PROGRAM P_MotionControl
VAR
	fbJoystick 				: FB_Joystick;
	fbGetStartPos 			: FB_StartPos;
	fbWinchVelIntegrator 	: FB_Integrator;
	fWinchVelRef 			: LREAL;
	fWinchPosRef 			: LREAL;
	fWinchPos 				: LREAL;
	fInitialWinchPos 		: LREAL;
	bWinchVelIntegratorOn	: BOOL := TRUE; 
	bAutoEnable 			: BOOL;
	bManualEnable 			: BOOL;
	fWinchPosRefManual 		: LREAL;
	fWinchVelRefManual 		: LREAL;
	fWinchVelRefAuto 		: LREAL;
END_VAR

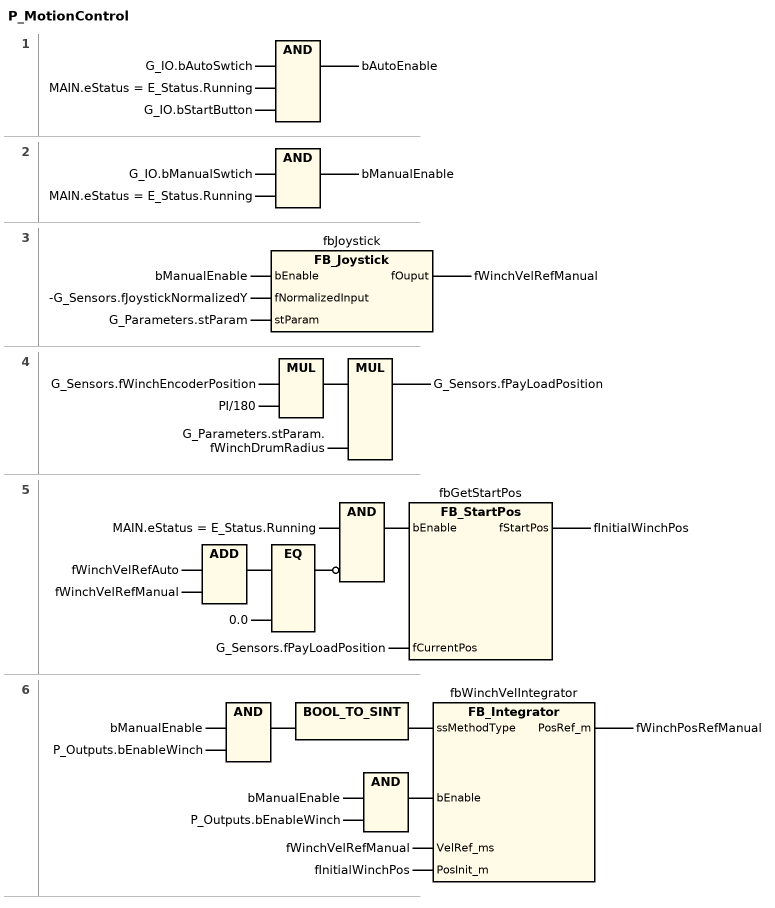
// NETWORK 1
bAutoEnable := G_IO.bAutoSwtich AND (MAIN.eStatus = E_Status.Running) AND G_IO.bStartButton;

// NETWORK 2
bManualEnable := G_IO.bManualSwtich AND (MAIN.eStatus = E_Status.Running);

// NETWORK 3
fbJoystick(
    bEnable := bManualEnable,
    fNormalizedInput := -G_Sensors.fJoystickNormalizedY,
    stParam := G_Parameters.stParam); // FB_Joystick
fWinchVelRefManual := fbJoystick.fOuput;

// NETWORK 4
G_Sensors.fPayLoadPosition := (G_Sensors.fWinchEncoderPosition * (PI/180)) * G_Parameters.stParam.fWinchDrumRadius;

// NETWORK 5
fbGetStartPos(bEnable := (MAIN.eStatus = E_Status.Running) AND NOT (fWinchVelRefAuto + fWinchVelRefManual = 0.0), fCurrentPos := G_Sensors.fPayLoadPosition); // FB_StartPos
fInitialWinchPos := fbGetStartPos.fStartPos;

// NETWORK 6
fbWinchVelIntegrator(
    ssMethodType := BOOL_TO_SINT(bManualEnable AND P_Outputs.bEnableWinch),
    bEnable := bManualEnable AND P_Outputs.bEnableWinch,
    VelRef_ms := fWinchVelRefManual,
    PosInit_m := fInitialWinchPos); // FB_Integrator
fWinchPosRefManual := fbWinchVelIntegrator.PosRef_m;

END_PROGRAM

(* stored: Version 1.1.0.1, ProductVersion 3.1.4026.11
   POU P_MotionControl: Id {fca9df39-4db4-416e-89b5-b1157c751beb}, SpecialFunc None *)
